PROGRAM MAIN
VAR
	ing1 AT %I* :BOOL;
	ing2 AT %I* :BOOL;
	ing3 AT %I* :BOOL;
	ing4 AT %I* :BOOL;
    uit1 AT%Q*:BOOL;
	uit2 AT%Q*:BOOL;
	uit3 AT%Q*:BOOL;
	uit4 AT%Q*:BOOL;
	
	
END_VAR


	uit1:= ing1;
	uit2:= ing1;
	uit3:= ing1;
	uit4:= ing1;

END_PROGRAM

(* stored: Version 1.1.0.1, ProductVersion 3.1.4022.11
   POU MAIN: Id {a4f99ad4-3d99-4cc3-aec6-4b8f25d45e95}, SpecialFunc None *)
